Yaskawa INFORM job: COMARC_TEST.JBI

/JOB
//NAME COMARC_TEST
//POS
///NPOS 4,4,0,0,0,0
///TOOL 0
///POSTYPE ROBOT
///RECTAN
///RCONF 1,0,0,0,0,0,0,0,0,0,0,0,0,0,0,0,0,0,0,0,0,0,0,0
C00000=377.304,12.750,-944.566,-0.0002,45.0020,-0.0063
C00001=395.380,64.109,-944.563,0.0000,45.0024,-0.0059
C00002=377.309,12.739,-951.129,-0.0005,45.0013,-0.0057
C00003=377.299,69.994,-951.127,0.0004,45.0019,-0.0032
///RCONF 0,0,0,0,0,0,0,0,0,0,0,0,0,0,0,0,0,0,0,0,0,0,0,0
BC00000=3036.073
BC00001=3036.073
BC00002=3036.073
BC00003=3036.073
//INST
///DATE 2024/10/23 15:24
///ATTR SC,RW,RJ
////FRAME ROBOT
///GROUP1 RB1,BS1
NOP
REFP 1 C00000 BC00000
REFP 2 C00001 BC00001
MACRO1 MJ#(0) ARGF50
MOVL C00002 BC00002 V=8.3 PL=0
ARCON
COMARCON AMP=0.5 FREQ=2.5 ANGL=45.0 U/D=4800 L/R=0.0
MOVL C00003 BC00003 V=8.3
ARCOF
COMARCOF
END
